SUBAPPLICATION DDS_CLIENT (* Wrapper for DDS Publisher and Subscriber Pair as a Client *)
  (* Standard: 61499-2 *)
  (* Version 1.0, 2023-03-15, Tim Hesse *)
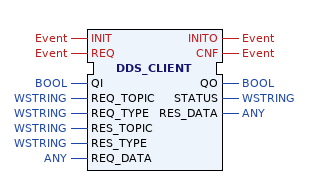
  EVENT_INPUT
    INIT; (* Initialization Request *)
    REQ; (* Normal Execution Request *)
  END_EVENT
  EVENT_OUTPUT
    INITO; (* Initialization Confirm *)
    CNF; (* Execution Confirmation *)
  END_EVENT
  VAR_INPUT
    QI : BOOL; (* Input event qualifier *)
    REQ_TOPIC : WSTRING; (* Request DDS Topic *)
    REQ_TYPE : WSTRING; (* Request DDS Type *)
    RES_TOPIC : WSTRING; (* Response DDS Topic *)
    RES_TYPE : WSTRING; (* Response DDS Type *)
    REQ_DATA : ANY; (* Request Data *)
  END_VAR
  VAR_OUTPUT
    QO : BOOL; (* Output event qualifier *)
    STATUS : WSTRING; (* Service Status *)
    RES_DATA : ANY; (* Response Data *)
  END_VAR
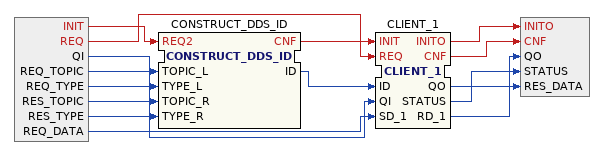
  FBS
    CONSTRUCT_DDS_ID : CONSTRUCT_DDS_ID;
    CLIENT_1 : CLIENT_1;
  END_FBS
  EVENT_CONNECTIONS
    CONSTRUCT_DDS_ID.CNF TO CLIENT_1.INIT;
    REQ TO CLIENT_1.REQ;
    CLIENT_1.INITO TO INITO;
    CLIENT_1.CNF TO CNF;
    INIT TO CONSTRUCT_DDS_ID.REQ2;
  END_CONNECTIONS
  DATA_CONNECTIONS
    REQ_TOPIC TO CONSTRUCT_DDS_ID.TOPIC_L;
    REQ_TYPE TO CONSTRUCT_DDS_ID.TYPE_L;
    CLIENT_1.QO TO QO;
    CLIENT_1.STATUS TO STATUS;
    CONSTRUCT_DDS_ID.ID TO CLIENT_1.ID;
    QI TO CLIENT_1.QI;
    REQ_DATA TO CLIENT_1.SD_1;
    RES_TOPIC TO CONSTRUCT_DDS_ID.TOPIC_R;
    RES_TYPE TO CONSTRUCT_DDS_ID.TYPE_R;
    CLIENT_1.RD_1 TO RES_DATA;
  END_CONNECTIONS
END_SUBAPPLICATION
